// TIA Portal V15.1 export
// export: Created 2024-06-21T08:40:49.022185Z, ExportSetting WithDefaults, DisplayName Totally Integrated Automation Portal, DisplayVersion V15.1 Update 5, DisplayName TIA Portal Openness, DisplayVersion V15.1 Update 5, DisplayName SINAMICS Startdrive Advanced, DisplayVersion V15.1, DisplayName G130, G150, S120, S150, SINAMICS MV, S210, DisplayVersion V15.1, DisplayName G110M, G120, G120C, G120D, G120P, DisplayVersion V15.1, DisplayName STEP 7 Professional, DisplayVersion V15.1 Update 5, DisplayName STEP 7 Safety, DisplayVersion V15.1, DisplayName WinCC Professional, DisplayVersion V15.1 Update 5, DisplayName SIMATIC Visualization Architect, DisplayVersion V15.1
DATA_BLOCK "_209220ZM01"   // DB350
{ S7_Optimized_Access := 'FALSE' }
AUTHOR : VCG
VERSION : 0.1
// stored: AutoNumber false, DBAccessibleFromOPCUA true, IsOnlyStoredInLoadMemory false, IsWriteProtectedInAS false
   VAR RETAIN
      AA_209220CS22M4SG40 { ExternalAccessible := 'False'; ExternalVisible := 'False'; ExternalWritable := 'False'} : Bool;   // Open Door Control NOK
      AA_209220CS22M4SG41 { ExternalAccessible := 'False'; ExternalVisible := 'False'; ExternalWritable := 'False'} : Bool;   // Open Door Control NOK
      AC_209220CS22M4SG40 { ExternalAccessible := 'False'; ExternalVisible := 'False'; ExternalWritable := 'False'} : Bool;   // Open Door Control disabled from HMI
      AC_209220CS22M4SG41 { ExternalAccessible := 'False'; ExternalVisible := 'False'; ExternalWritable := 'False'} : Bool;   // Open Door Control disabled from HMI
      AC_209220CHB21M14SG2 { ExternalAccessible := 'False'; ExternalVisible := 'False'; ExternalWritable := 'False'} : Bool;   // Detection OK to close Holdback NOK
      AC_BodyCounterConv1 { ExternalAccessible := 'False'; ExternalVisible := 'False'; ExternalWritable := 'False'} : Bool;   // Body Counter below 0 or above MAX
      AlarmA { ExternalAccessible := 'False'; ExternalVisible := 'False'; ExternalWritable := 'False'} : Bool;   // Summary Alarm A
      AlarmB { ExternalAccessible := 'False'; ExternalVisible := 'False'; ExternalWritable := 'False'} : Bool;   // Summary Alarm B
      AlarmC { ExternalAccessible := 'False'; ExternalVisible := 'False'; ExternalWritable := 'False'} : Bool;   // Summary Alarm C
      AlarmD { ExternalAccessible := 'False'; ExternalVisible := 'False'; ExternalWritable := 'False'} : Bool;   // Summary Alarm D
      AlarmABCondition { ExternalAccessible := 'False'; ExternalVisible := 'False'; ExternalWritable := 'False'} : Bool;   // Alarm AB condition
      ZMS011AlarmA { ExternalAccessible := 'False'; ExternalVisible := 'False'; ExternalWritable := 'False'} : Bool;   // Summary Alarm A
      ZMS011AlarmB { ExternalAccessible := 'False'; ExternalVisible := 'False'; ExternalWritable := 'False'} : Bool;   // Summary Alarm B
      ZMS011AlarmC { ExternalAccessible := 'False'; ExternalVisible := 'False'; ExternalWritable := 'False'} : Bool;   // Summary Alarm C
      ZMS011AlarmD { ExternalAccessible := 'False'; ExternalVisible := 'False'; ExternalWritable := 'False'} : Bool;   // Summary Alarm D
      ZMS011AlarmABCondition { ExternalAccessible := 'False'; ExternalVisible := 'False'; ExternalWritable := 'False'} : Bool;   // Alarm AB condition
      ZMS012AlarmA { ExternalAccessible := 'False'; ExternalVisible := 'False'; ExternalWritable := 'False'} : Bool;   // Summary Alarm A
      ZMS012AlarmB { ExternalAccessible := 'False'; ExternalVisible := 'False'; ExternalWritable := 'False'} : Bool;   // Summary Alarm B
      ZMS012AlarmC { ExternalAccessible := 'False'; ExternalVisible := 'False'; ExternalWritable := 'False'} : Bool;   // Summary Alarm C
      ZMS012AlarmD { ExternalAccessible := 'False'; ExternalVisible := 'False'; ExternalWritable := 'False'} : Bool;   // Summary Alarm D
      ZMS012AlarmABCondition { ExternalAccessible := 'False'; ExternalVisible := 'False'; ExternalWritable := 'False'} : Bool;   // Alarm AB condition
      ZMS013AlarmA { ExternalAccessible := 'False'; ExternalVisible := 'False'; ExternalWritable := 'False'} : Bool;   // Summary Alarm A
      ZMS013AlarmB { ExternalAccessible := 'False'; ExternalVisible := 'False'; ExternalWritable := 'False'} : Bool;   // Summary Alarm B
      ZMS013AlarmC { ExternalAccessible := 'False'; ExternalVisible := 'False'; ExternalWritable := 'False'} : Bool;   // Summary Alarm C
      ZMS013AlarmD { ExternalAccessible := 'False'; ExternalVisible := 'False'; ExternalWritable := 'False'} : Bool;   // Summary Alarm D
      ZMS013AlarmABCondition { ExternalAccessible := 'False'; ExternalVisible := 'False'; ExternalWritable := 'False'} : Bool;   // Alarm AB condition
      H_Anim : Word;   // Animation
      H_DBnr : Int;   // DB number
      H_HMICmd : Word;   // HMI Command
      H_OrdersIAnim : DWord;   // HMI Animation of the icon
      H_DataHandlingIAnim : Word;   // HMI Animation of the icon
      H_AndonIAnim : Word;   // HMI Animation of the icon
      H_Counter1WeekIAnim : Word;   // HMI Animation of the icon
      H_209220CHB21M14SG2IAnim : DWord;   // HMI Animation of the icon
      H_209220CS22M4SG40IAnim : DWord;   // HMI Animation of the icon
      H_209220CS22M4SG41IAnim : DWord;   // HMI Animation of the icon
      H_HMI : Struct   // Icon Animation
         BodyCounter : "H_HMI";   // HMI Animation of the icon
         CRClockStartStop : "H_HMI";   // HMI Animation of the icon
         "209220CS22ShiftRegLine" : "H_HMI";   // HMI Animation of the icon
         "209220CS22ProdSpeed" : "H_HMI";   // HMI Animation of the icon
         "209220CS22LineFeed" : "H_HMI";   // HMI Animation of the icon
         "209220CS22ProdStartStop" : "H_HMI";   // HMI Animation of the icon
         "209220CHB21" : "H_HMI";   // HMI Animation of the icon
         "209220CR21" : "H_HMI";   // HMI Animation of the icon
         "209220CS22" : "H_HMI";   // HMI Animation of the icon
         "209220CR23" : "H_HMI";   // HMI Animation of the icon
      END_STRUCT;
      H : Struct   // Animation
         BodyCounter : "H_GBBodyCounter";   // HMI Animation
         CRClockStartStop : "H_GBCRClockStartStop";   // HMI Animation
         "209220CS22ShiftRegLine" : "H_GBShiftRegLine";   // HMI Animation
         "209220CS22ProdSpeed" : "H_GBProdSpeed";   // HMI Animation
         "209220CS22LineFeed" : "H_GBLineFeed";   // HMI Animation
         "209220CS22ProdStartStop" : "H_GBProdStartStop";   // HMI Animation
         "209220CS22ProdInfo" : "H_GBProdInfo";   // HMI Animation
         "209220CHB21" : "H_GBMovUnit2Pos2W2S-MoviFitFCPN";   // HMI Animation
         "209220CR21" : "H_GBRoller2W2S-MDXPN-6PD-DFS22B";   // HMI Animation
         "209220CS22" : "H_GBLineConvBrake-MDXPN-DFS22B";   // HMI Animation
         "209220CR23" : "H_GBRoller2W2S-MDXPN-6PD-DFS22B";   // HMI Animation
      END_STRUCT;
      H_209220ZMS011IAnim : Word;   // 209220ZMS011: For animation of icon
      H_209220ZMS012IAnim : Word;   // 209220ZMS012: For animation of icon
      H_209220ZMS013IAnim : Word;   // 209220ZMS013: For animation of icon
      H_308220ZM01IAnim : Word;   // 308220ZM01: For animation of icon
      H_212AIAnim : Word;   // 212A: For animation of icon
      "209220CHB21" { ExternalAccessible := 'False'; ExternalVisible := 'False'; ExternalWritable := 'False'} : "MovUnit";   // HoldBack
      "209220CR21" { ExternalAccessible := 'False'; ExternalVisible := 'False'; ExternalWritable := 'False'} : "Conveyor";   // Roller
      "209220CS22" { ExternalAccessible := 'False'; ExternalVisible := 'False'; ExternalWritable := 'False'} : "LineConv";   // Line Conveyor
      "209220CR23" { ExternalAccessible := 'False'; ExternalVisible := 'False'; ExternalWritable := 'False'} : "Conveyor";   // Roller
      "209220ZMS011" { ExternalAccessible := 'False'; ExternalVisible := 'False'; ExternalWritable := 'False'} : "AlarmBits";   // Mode Alarm Bits
      "209220ZMS012" { ExternalAccessible := 'False'; ExternalVisible := 'False'; ExternalWritable := 'False'} : "AlarmBits";   // Mode Alarm Bits
      "209220ZMS013" { ExternalAccessible := 'False'; ExternalVisible := 'False'; ExternalWritable := 'False'} : "AlarmBits";   // Mode Alarm Bits
      Orders { ExternalAccessible := 'False'; ExternalVisible := 'False'; ExternalWritable := 'False'} : "AlarmBits";   // Orders Alarm Bits
      DataHandling { ExternalAccessible := 'False'; ExternalVisible := 'False'; ExternalWritable := 'False'} : "AlarmBits";   // DataHandling Alarm Bits
      Andon { ExternalAccessible := 'False'; ExternalVisible := 'False'; ExternalWritable := 'False'} : "AlarmBits";   // Andon Alarm Bits
      BodyCounter { ExternalAccessible := 'False'; ExternalVisible := 'False'; ExternalWritable := 'False'} : "BodyCounter";   // Body Counter
      SumModes { ExternalAccessible := 'False'; ExternalVisible := 'False'; ExternalWritable := 'False'} : "Modes";   // Summary Modes
      HomePosition { ExternalAccessible := 'False'; ExternalVisible := 'False'; ExternalWritable := 'False'} : Bool;   // Home position
      EmptyStnReached { ExternalAccessible := 'False'; ExternalVisible := 'False'; ExternalWritable := 'False'} : Bool;   // Empty Station is Reached
      SumAutoMode { ExternalAccessible := 'False'; ExternalVisible := 'False'; ExternalWritable := 'False'} : Bool;   // Summary Auto Mode in safety zone
      SumAutoModeSel { ExternalAccessible := 'False'; ExternalVisible := 'False'; ExternalWritable := 'False'} : Bool;   // Summary Auto Mode Select in safety zone
      SumStepMode { ExternalAccessible := 'False'; ExternalVisible := 'False'; ExternalWritable := 'False'} : Bool;   // Summary Step Mode in safety zone
      SumStepModeSel { ExternalAccessible := 'False'; ExternalVisible := 'False'; ExternalWritable := 'False'} : Bool;   // Summary Step Mode Select in safety zone
      SumHomeRunMode { ExternalAccessible := 'False'; ExternalVisible := 'False'; ExternalWritable := 'False'} : Bool;   // Summary Home Run Mode in safety zone
      SumHomerunModeSel { ExternalAccessible := 'False'; ExternalVisible := 'False'; ExternalWritable := 'False'} : Bool;   // Summary Home Run Mode Select in safety zone
      SumManualMode { ExternalAccessible := 'False'; ExternalVisible := 'False'; ExternalWritable := 'False'} : Bool;   // Summary Manual Mode in safety zone
      SumManualModeSel { ExternalAccessible := 'False'; ExternalVisible := 'False'; ExternalWritable := 'False'} : Bool;   // Summary Manual Mode Select in safety zone
      SumAnyProdModeActive { ExternalAccessible := 'False'; ExternalVisible := 'False'; ExternalWritable := 'False'} : Bool;   // Summary Any Production Mode Active in safety zone
      SumAnyProdModeSel { ExternalAccessible := 'False'; ExternalVisible := 'False'; ExternalWritable := 'False'} : Bool;   // Summary Any Production Mode Select in safety zone
      "220CS22ReadyForOperation" { ExternalAccessible := 'False'; ExternalVisible := 'False'; ExternalWritable := 'False'} : Bool;   // Drive Ready For Operation
      "220CS22Saturation" { ExternalAccessible := 'False'; ExternalVisible := 'False'; ExternalWritable := 'False'} : Bool;   // Saturation
      "220CS22EcoMode" { ExternalAccessible := 'False'; ExternalVisible := 'False'; ExternalWritable := 'False'} : Bool;   // Eco Mode
      "220CHB21M14SG2CheckOn" { ExternalAccessible := 'False'; ExternalVisible := 'False'; ExternalWritable := 'False'} : Bool;   // Check On OK to close Holdback
      "220CHB21M14SG2DetOn" { ExternalAccessible := 'False'; ExternalVisible := 'False'; ExternalWritable := 'False'} : Bool;   // OK to close Holdback
      "220CS22M4SG4xZoneCheckOn" { ExternalAccessible := 'False'; ExternalVisible := 'False'; ExternalWritable := 'False'} : Bool;   // Zone Check On Open Door Control
      "220CS22M4SG40AlarmABCondition" { ExternalAccessible := 'False'; ExternalVisible := 'False'; ExternalWritable := 'False'} : Bool;   // Alarm AB Condition
      "220CS22M4SG40CheckOn" { ExternalAccessible := 'False'; ExternalVisible := 'False'; ExternalWritable := 'False'} : Bool;   // Check On Open Door Control
      "220CS22M4SG40DetOn" { ExternalAccessible := 'False'; ExternalVisible := 'False'; ExternalWritable := 'False'} : Bool;   // Open Door Control On
      "220CS22M4SG41AlarmABCondition" { ExternalAccessible := 'False'; ExternalVisible := 'False'; ExternalWritable := 'False'} : Bool;   // Alarm AB Condition
      "220CS22M4SG41CheckOn" { ExternalAccessible := 'False'; ExternalVisible := 'False'; ExternalWritable := 'False'} : Bool;   // Check On Open Door Control
      "220CS22M4SG41DetOn" { ExternalAccessible := 'False'; ExternalVisible := 'False'; ExternalWritable := 'False'} : Bool;   // Open Door Control On
      "______Production Line__________________" { ExternalAccessible := 'False'; ExternalVisible := 'False'; ExternalWritable := 'False'} : Bool;   // --------------------------------------------------------------------------------
      "209220ZM01CRClockStartStop" { ExternalAccessible := 'False'; ExternalVisible := 'False'; ExternalWritable := 'False'} : "CRClockStartStop";   // Production Line - Clock Control Room
      "209220CS22ProdSpeed" { ExternalAccessible := 'False'; ExternalVisible := 'False'; ExternalWritable := 'False'} : "ProdSpeed";   // Production Line - Production Speed
      "209220CS22LineFeed" { ExternalAccessible := 'False'; ExternalVisible := 'False'; ExternalWritable := 'False'} : "LineFeed";   // Production Line - Line Feed
      "209220CS22ProdStartStop" { ExternalAccessible := 'False'; ExternalVisible := 'False'; ExternalWritable := 'False'} : "ProdStartStop";   // Production Line - Production Start Stop
      "209220CS22ShiftRegLine" { ExternalAccessible := 'False'; ExternalVisible := 'False'; ExternalWritable := 'False'} : "ShiftRegLine";   // Production Line - Shift Register
      "209220CS22ShiftRegData" { ExternalAccessible := 'False'; ExternalVisible := 'False'; ExternalWritable := 'False'} : "ShiftRegData";   // Production Line - Shift Register Line data
      "209220CS22ShiftRegTriggerDetection" { ExternalAccessible := 'False'; ExternalVisible := 'False'; ExternalWritable := 'False'} : Bool;   // Production Line - Shift Register Trigger detection
      "209220CS22ShiftRegPartPresent" { ExternalAccessible := 'False'; ExternalVisible := 'False'; ExternalWritable := 'False'} : Bool;   // Production Line - Part present in Shiftregister
      Edge { ExternalAccessible := 'False'; ExternalVisible := 'False'; ExternalWritable := 'False'} : Array[1..10] of Bool;   // Edge
   END_VAR
BEGIN
END_DATA_BLOCK
